Staubli VAL3: moveNext.pgx

program moveNext()
begin
  currentSamPosJ=herej()
  currentSamPos=jointToPoint(flange,world,currentSamPosJ)
  movel(appro(currentSamPos,{(numXarray-1)*-17.03,(numYarray-1)*-17,0,0,0,0}),flange,mFastMov)
  waitEndMove()
end
